// TIA Portal project "practica 1" (V18)

(* hardware
DEVICE "S7-300/ET200M station_1"  S7-300 station
   slot 0: "Rail_0"  Rail  6ES7 390-1***0-0AA0
   slot 2: "PLC_1"  CPU 313C-2 DP  6ES7 313-6CF03-0AB0  V2.6
      slot 0: "MPI interface_1"  X1
      slot 1: "DP interface_1"  X2
      slot 2: "DI 16/DO 16_1"  DI16/DO16
      slot 4: "Count_1"  Counter
*)

// ===== PLC "PLC_1"  CPU 313C-2 DP =====

VAR_GLOBAL   // PLC tag table "Default tag table"
   "A" AT %MD1 : Real;   // Coeficiente cuadrático
   "B" AT %MD5 : Real;   // Coeficiente lineal
   "C" AT %MD10 : Real;   // Término independiente
   "Discriminante" AT %MD15 : Real;   // B² - 4AC
   "Raiz" AT %MD20 : Real;   // √Discriminante
   "Numerador" AT %MD25 : Real;   // -B + Raiz
   "Denominador" AT %MD30 : Real;   // 2A
   "Resultado" AT %MD35 : Real;   // Resultado final
   "ResultadoRedondeado" AT %MD40 : DInt;   // Resultado redondeado a entero
   "ResultadoWORD" AT %QW124 : Word;   // Resultado para QW124 (en binario)
   "BotonA_Anterior" AT %M0.0 : Bool;   // Estado anterior de botón A
   "BotonB_Anterior" AT %M0.1 : Bool;   // Estado anterior de botón B
   "BotonC_Anterior" AT %M0.2 : Bool;   // Estado anterior de botón C
   "Pulsado_A" AT %M0.3 : Bool;   // Flanco positivo A
   "Pulsado_B" AT %M0.4 : Bool;   // Flanco positivo B
   "Pulsado_C" AT %M0.5 : Bool;   // Flanco positivo C
   "Boton_A" AT %I125.2 : Bool;   // Botón para A
   "Boton_B" AT %I125.3 : Bool;   // Botón para B
   "Boton_C" AT %I125.4 : Bool;   // Botón para C
   "TMP1" AT %MD45 : Real;
   "TMP2" AT %MD50 : Real;
   "TMP3" AT %MD55 : Real;
   "TMP4" AT %MD60 : Real;
END_VAR

FUNCTION "Block_1" : Void   // FC1, LAD
{ S7_Optimized_Access := 'FALSE' }
VERSION : 0.1
   VAR_INPUT
      "A" : Bool;
      "B" : Bool;
      C : Bool;
   END_VAR
   VAR_OUTPUT
      "Resultdo X1" : Word;
      a_1 : Real;
      b_1 : Real;
      c_1 : Real;
   END_VAR
BEGIN

REGION Network 1: Flanco positivo A
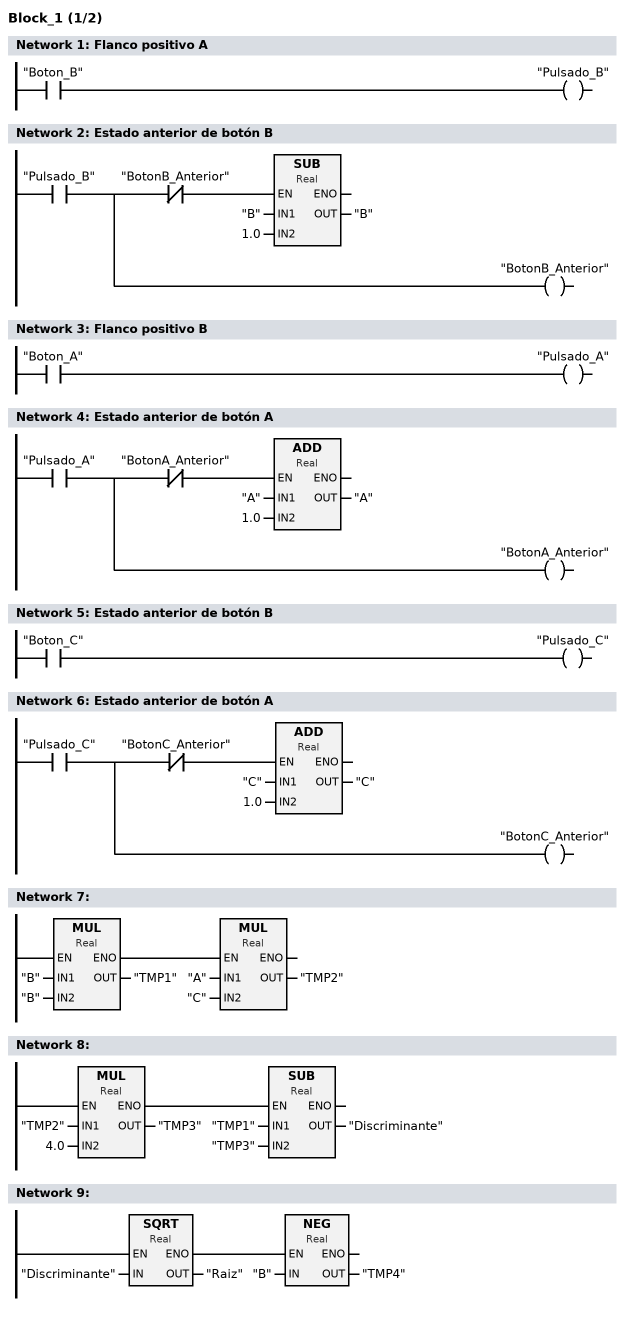
   RUNG wire#powerrail
      Contact( "Boton_B" )
      Coil( "Pulsado_B" )
   END_RUNG
   // the same network as SCL:
   "Pulsado_B" := "Boton_B";
END_REGION

REGION Network 2: Estado anterior de botón B
   RUNG wire#powerrail
      Contact( "Pulsado_B" )
      wire#w1
      I_Contact( "BotonB_Anterior" )
      { S7_Templates := "SrcType := Real"; S7_GenerateENO := "TRUE" } Sub(in1 := "B", in2 := 1.0, out => "B")
   END_RUNG
   RUNG wire#w1
      Coil( "BotonB_Anterior" )
   END_RUNG
   // the same network as SCL:
   IF "Pulsado_B" AND NOT "BotonB_Anterior" THEN "B" := "B" - 1.0; END_IF;
   "BotonB_Anterior" := "Pulsado_B";
END_REGION

REGION Network 3: Flanco positivo B
   RUNG wire#powerrail
      Contact( "Boton_A" )
      Coil( "Pulsado_A" )
   END_RUNG
   // the same network as SCL:
   "Pulsado_A" := "Boton_A";
END_REGION

REGION Network 4: Estado anterior de botón A
   RUNG wire#powerrail
      Contact( "Pulsado_A" )
      wire#w1
      I_Contact( "BotonA_Anterior" )
      { S7_Templates := "SrcType := Real"; S7_GenerateENO := "TRUE" } Add(in1 := "A", in2 := 1.0, out => "A")
   END_RUNG
   RUNG wire#w1
      Coil( "BotonA_Anterior" )
   END_RUNG
   // the same network as SCL:
   IF "Pulsado_A" AND NOT "BotonA_Anterior" THEN "A" := "A" + 1.0; END_IF;
   "BotonA_Anterior" := "Pulsado_A";
END_REGION

REGION Network 5: Estado anterior de botón B
   RUNG wire#powerrail
      Contact( "Boton_C" )
      Coil( "Pulsado_C" )
   END_RUNG
   // the same network as SCL:
   "Pulsado_C" := "Boton_C";
END_REGION

REGION Network 6: Estado anterior de botón A
   RUNG wire#powerrail
      Contact( "Pulsado_C" )
      wire#w1
      I_Contact( "BotonC_Anterior" )
      { S7_Templates := "SrcType := Real"; S7_GenerateENO := "TRUE" } Add(in1 := "C", in2 := 1.0, out => "C")
   END_RUNG
   RUNG wire#w1
      Coil( "BotonC_Anterior" )
   END_RUNG
   // the same network as SCL:
   IF "Pulsado_C" AND NOT "BotonC_Anterior" THEN "C" := "C" + 1.0; END_IF;
   "BotonC_Anterior" := "Pulsado_C";
END_REGION

REGION Network 7
   RUNG wire#powerrail
      { S7_Templates := "SrcType := Real"; S7_GenerateENO := "TRUE" } Mul(in1 := "B", in2 := "B", out => "TMP1")
      { S7_Templates := "SrcType := Real"; S7_GenerateENO := "TRUE" } Mul(in1 := "A", in2 := "C", out => "TMP2")
   END_RUNG
   // the same network as SCL:
   // ENO of a box is taken as its EN; it also drops when the box reports an error
   "TMP1" := "B" * "B";
   "TMP2" := "A" * "C";
END_REGION

REGION Network 8
   RUNG wire#powerrail
      { S7_Templates := "SrcType := Real"; S7_GenerateENO := "TRUE" } Mul(in1 := "TMP2", in2 := 4.0, out => "TMP3")
      { S7_Templates := "SrcType := Real"; S7_GenerateENO := "TRUE" } Sub(in1 := "TMP1", in2 := "TMP3", out => "Discriminante")
   END_RUNG
   // the same network as SCL:
   // ENO of a box is taken as its EN; it also drops when the box reports an error
   "TMP3" := "TMP2" * 4.0;
   "Discriminante" := "TMP1" - "TMP3";
END_REGION

REGION Network 9
   // ENO of a box is taken as its EN; it also drops when the box reports an error
   "Raiz" := SQRT("Discriminante");
   "TMP4" := -"B";
END_REGION

REGION Network 10
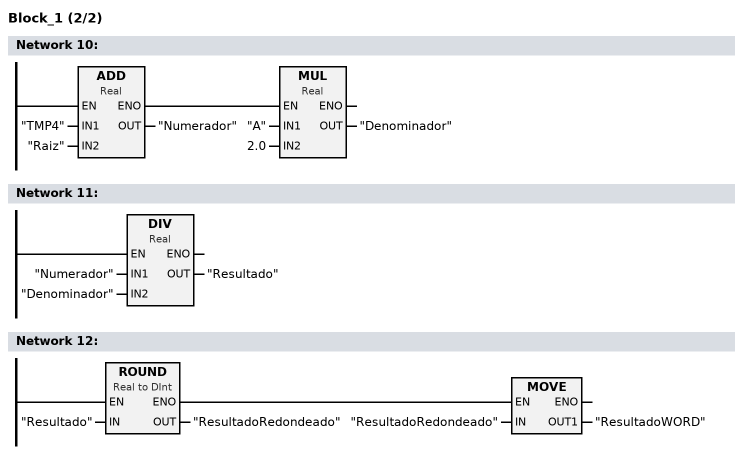
   RUNG wire#powerrail
      { S7_Templates := "SrcType := Real"; S7_GenerateENO := "TRUE" } Add(in1 := "TMP4", in2 := "Raiz", out => "Numerador")
      { S7_Templates := "SrcType := Real"; S7_GenerateENO := "TRUE" } Mul(in1 := "A", in2 := 2.0, out => "Denominador")
   END_RUNG
   // the same network as SCL:
   // ENO of a box is taken as its EN; it also drops when the box reports an error
   "Numerador" := "TMP4" + "Raiz";
   "Denominador" := "A" * 2.0;
END_REGION

REGION Network 11
   RUNG wire#powerrail
      { S7_Templates := "SrcType := Real"; S7_GenerateENO := "TRUE" } Div(in1 := "Numerador", in2 := "Denominador", out => "Resultado")
   END_RUNG
   // the same network as SCL:
   "Resultado" := "Numerador" / "Denominador";
END_REGION

REGION Network 12
   RUNG wire#powerrail
      { S7_Templates := "[SrcType := Real, DestType := DInt]"; S7_GenerateENO := "TRUE" } Round(in := "Resultado", out => "ResultadoRedondeado")
      { S7_GenerateENO := "TRUE" } Move(in := "ResultadoRedondeado", out1 => "ResultadoWORD")
   END_RUNG
   // the same network as SCL:
   // ENO of a box is taken as its EN; it also drops when the box reports an error
   "ResultadoRedondeado" := ROUND("Resultado");
   "ResultadoWORD" := "ResultadoRedondeado";
END_REGION
END_FUNCTION

ORGANIZATION_BLOCK "Main"   // OB1, LAD
TITLE = "Main Program Sweep (Cycle)"
{ S7_Optimized_Access := 'FALSE' }
VERSION : 0.1
   VAR_TEMP
      OB1_EV_CLASS : Byte;   // Bits 0-3 = 1 (Coming event), Bits 4-7 = 1 (Event class 1)
      OB1_SCAN_1 : Byte;   // 1 (Cold restart scan 1 of OB 1), 3 (Scan 2-n of OB 1)
      OB1_PRIORITY : Byte;   // Priority of OB Execution
      OB1_OB_NUMBR : Byte;   // 1 (Organization block 1, OB1)
      OB1_RESERVED_1 : Byte;   // Reserved for system
      OB1_RESERVED_2 : Byte;   // Reserved for system
      OB1_PREV_CYCLE : Int;   // Cycle time of previous OB1 scan (milliseconds)
      OB1_MIN_CYCLE : Int;   // Minimum cycle time of OB1 (milliseconds)
      OB1_MAX_CYCLE : Int;   // Maximum cycle time of OB1 (milliseconds)
      OB1_DATE_TIME : Date_And_Time;   // Date and time OB1 started
   END_VAR
BEGIN

REGION Network 1
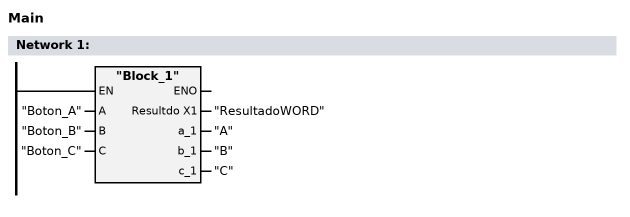
   RUNG wire#powerrail
      "Block_1"("A" := "Boton_A", "B" := "Boton_B", C := "Boton_C", "Resultdo X1" => "ResultadoWORD", a_1 => "A", b_1 => "B", c_1 => "C")
   END_RUNG
   // the same network as SCL:
   "Block_1"("A" := "Boton_A",
             "B" := "Boton_B",
             C := "Boton_C",
             "Resultdo X1" => "ResultadoWORD",
             a_1 => "A",
             b_1 => "B",
             c_1 => "C");
END_REGION
END_ORGANIZATION_BLOCK